// TIA Portal V20 export
TYPE "HMI_ILck8x4L"
   STRUCT
      In01_Text : String[16];   // In01 text
      BypIn : Word;   // Bypass In01 - In16 (via operator)
      AV01 : Real;   // Analog value for In01
      AV01_Unit : Int;   // Engineering unit of AV01
      In02_Text : String[16];   // In02 text
      AV02 : Real;   // Analog value for In02
      AV02_Unit : Int;   // Engineering unit of AV02
      In03_Text : String[16];   // In03 text
      AV03 : Real;   // Analog value for In03
      AV03_Unit : Int;   // Engineering unit of AV03
      In04_Text : String[16];   // In04 text
      AV04 : Real;   // Analog value for In04
      AV04_Unit : Int;   // Engineering unit of AV04
      In05_Text : String[16];   // In05 text
      AV05 : Real;   // Analog value for In05
      AV05_Unit : Int;   // Engineering unit of AV05
      In06_Text : String[16];   // In06 text
      AV06 : Real;   // Analog value for In06
      AV06_Unit : Int;   // Engineering unit of AV06
      In07_Text : String[16];   // In07 text
      AV07 : Real;   // Analog value for In07
      AV07_Unit : Int;   // Engineering unit of AV07
      In08_Text : String[16];   // In08 text
      AV08 : Real;   // Analog value for In08
      AV08_Unit : Int;   // Engineering unit of AV08
      In09_Text : String[16];   // In09 text
      AV09 : Real;   // Analog value for In09
      AV09_Unit : Int;   // Engineering unit of AV09
      In10_Text : String[16];   // In10 text
      AV10 : Real;   // Analog value for In10
      AV10_Unit : Int;   // Engineering unit of AV10
      In11_Text : String[16];   // In11 text
      AV11 : Real;   // Analog value for In11
      AV11_Unit : Int;   // Engineering unit of AV11
      In12_Text : String[16];   // In12 text
      AV12 : Real;   // Analog value for In12
      AV12_Unit : Int;   // Engineering unit of AV12
      In13_Text : String[16];   // In13 text
      AV13 : Real;   // Analog value for In13
      AV13_Unit : Int;   // Engineering unit of AV13
      In14_Text : String[16];   // In14 text
      AV14 : Real;   // Analog value for In14
      AV14_Unit : Int;   // Engineering unit of AV14
      In15_Text : String[16];   // In15 text
      AV15 : Real;   // Analog value for In15
      AV15_Unit : Int;   // Engineering unit of AV15
      In16_Text : String[16];   // In16 text
      AV16 : Real;   // Analog value for In16
      AV16_Unit : Int;   // Engineering unit of AV16
      BypOp : DWord;   // Temp. Bypass by operator In01 - In16, Out
      BypTime : Real := 30.0;   // Temp. Bypass TIME[s]
      BypPreWarnTime : Real := 10.0;   // Temp. Bypass prewarning TIME[s]
      BypRST : Bool;   // Temp. Bypass Restart
      RstOp : Bool;   // Reset Interlock by operator
      Out_Byp : Bool;   // Bypass by operator
      RstFirstOp : Bool;   // Reset FirstIn (operator)
      RstBypOp : Bool;   // Reset all Bypasses (Operator)
      ILckTime : Real;   // Time on-/off delay or timed Interlock[s]
      BypTime_Out { ExternalWritable := 'False'} : Real;   // Temp. Bypass time left
      ILckTime_Out { ExternalWritable := 'False'} : Real;   // Interlock time left
      OS_PermOut { ExternalWritable := 'False'} : DWord := DWORD#16#FFFF_FFFF;   // Operator Permission: Output for OS
      OS_PermLog { ExternalWritable := 'False'} : DWord := DWORD#16#FFFF_FFFF;   // Operator Permission: Output for OS
      OpSt_Out { ExternalWritable := 'False'} : DWord;   // Enabled operator stations
      TimeMode { ExternalWritable := 'False'} : Int;   // 0: No delay, 1: off delay, 2: on delay, 3: timed (Off), 4: timed (On)
      ST_Worst { ExternalWritable := 'False'} : Byte := BYTE#16#80;   // Worst Signal Status
      Out_Word { ExternalWritable := 'False'} : Word;   // Output(Output,Stage 1 - Stage 3)
      AV01_04_ST { ExternalWritable := 'False'} : DWord := DWORD#16#FFFF_FFFF;   // Analog value Signal Status for In01 - In04
      AV05_08_ST { ExternalWritable := 'False'} : DWord := DWORD#16#FFFF_FFFF;   // Analog value Signal Status for In05 - In08
      AV09_12_ST { ExternalWritable := 'False'} : DWord := DWORD#16#FFFF_FFFF;   // Analog value Signal Status for In09 - In12
      AV13_16_ST { ExternalWritable := 'False'} : DWord := DWORD#16#FFFF_FFFF;   // Analog value Signal Status for In13 - In16
      In01_04_ST { ExternalWritable := 'False'} : DWord := DWORD#16#FFFF_FFFF;   // Signal Status for In01 - In04
      In05_08_ST { ExternalWritable := 'False'} : DWord := DWORD#16#FFFF_FFFF;   // Signal Status for In05 - In08
      In09_12_ST { ExternalWritable := 'False'} : DWord := DWORD#16#FFFF_FFFF;   // Signal Status for In09 - In12
      In13_16_ST { ExternalWritable := 'False'} : DWord := DWORD#16#FFFF_FFFF;   // Signal Status for In13 -In16
      Out_ST { ExternalWritable := 'False'} : Byte := BYTE#16#FF;   // Output Signal Status
      Status1 { ExternalWritable := 'False'} : DWord;   // Status1
      Status2 { ExternalWritable := 'False'} : DWord;   // Status2
      Status3 { ExternalWritable := 'False'} : DWord;   // Status3
      Status4 { ExternalWritable := 'False'} : DWord;   // Status4
      Status5 { ExternalWritable := 'False'} : DWord;   // Status5
      Status6 { ExternalWritable := 'False'} : DWord;   // Status6
      Status7 { ExternalWritable := 'False'} : DWord;   // Status7
      Status8 { ExternalWritable := 'False'} : DWord;   // Status8
      Status9 { ExternalWritable := 'False'} : DWord;   // Status9
      Status10 { ExternalWritable := 'False'} : DWord;   // Status10
      Status11 { ExternalWritable := 'False'} : DWord;   // Status11
      Status12 { ExternalWritable := 'False'} : DWord;   // Status12
      Status13 { ExternalWritable := 'False'} : DWord;   // Status13
      Status14 { ExternalWritable := 'False'} : DWord;   // Status14
      Status15 { ExternalWritable := 'False'} : DWord;   // Status15
   END_STRUCT;
END_TYPE
